ABB RobotStudio station: RobotStudio.rsstnx

Station RobotStudio (saved by RobotStudio 23.3.10550.0)
Controller IRB120_3_58
  mechanical unit ROB_1: IRB120_3_58__01, 6 joints, base frame (0, 0, 0) mm
Layout (positions relative to the parent item):
  - IRB120_3_58__01 [mechanism, from %ABB.RobotStudio.Models.IRB120%\IRB120_3_58_G_01.rslib] at (0, 0, 0) mm; joint values [-0.8423, -0.388, 0.2778, -0.7289, 1.2738, -0.2663] (rad or m)
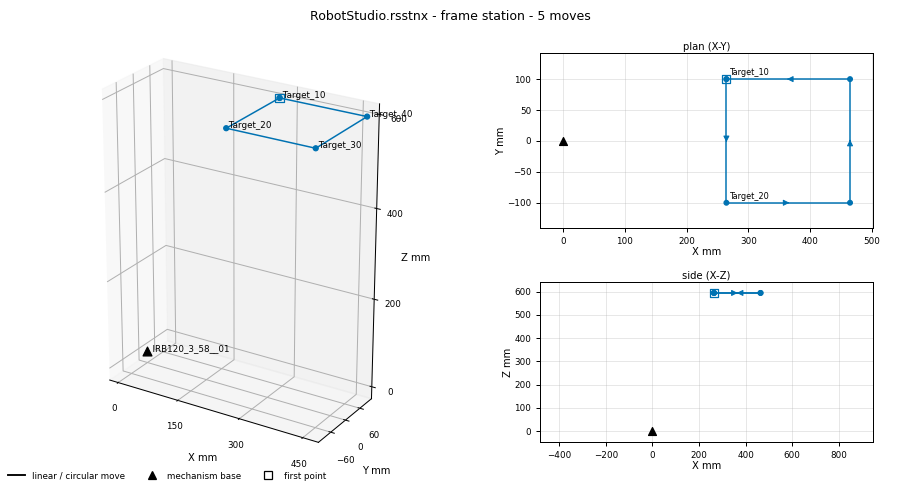
[picture p0: tool path of RobotStudio.rsstnx in frame station, 5 of 5 moves have a stored position in this frame; points joined in program order, loops and branches not executed]
Targets, tools, work objects and paths stored in the station, written as RAPID:
! task T_ROB1
MODULE MainModule
  CONST robtarget Target_10:=[[264.350012476,100.000011179,593.999948019],[0.500000001,0.000000007,0.866025403,0],[0,-1,0,0],[9E+09,9E+09,9E+09,9E+09,9E+09,9E+09]];
  CONST robtarget Target_20:=[[264.350012476,-100.000011179,593.999948019],[0.500000001,-0.000000007,0.866025403,0],[-1,0,-1,0],[9E+09,9E+09,9E+09,9E+09,9E+09,9E+09]];
  CONST robtarget Target_30:=[[464.350000726,-100.00000079,593.999945781],[0.500000003,-0.000000003,0.866025402,0.000000005],[-1,0,-1,0],[9E+09,9E+09,9E+09,9E+09,9E+09,9E+09]];
  CONST robtarget Target_40:=[[464.350000726,100.00000079,593.999945781],[0.500000003,0.000000003,0.866025402,-0.000000005],[0,-1,0,0],[9E+09,9E+09,9E+09,9E+09,9E+09,9E+09]];
  CONST robtarget Target_50:=[[264.350012476,100.000011179,593.999948019],[0.500000001,0.000000007,0.866025403,0],[0,-1,0,0],[9E+09,9E+09,9E+09,9E+09,9E+09,9E+09]];
  PROC Path_10()
    MoveJ Target_10,v400,z50,tool0\WObj:=wobj0;
    MoveL Target_20,v100,z50,tool0\WObj:=wobj0;
    MoveL Target_30,v100,z50,tool0\WObj:=wobj0;
    MoveL Target_40,v100,z50,tool0\WObj:=wobj0;
    MoveL Target_50,v100,z50,tool0\WObj:=wobj0;
  ENDPROC
  PROC main()
  ENDPROC
ENDMODULE

